TYPE ST_HIERARCHYDATALIST :
STRUCT
	TRACKINGLEVELS		:STRING;
	HIERARCHYDATAPK		:STRING;
	HIERARCHYDATAOUT	:STRING;
	HIERARCHYDATACS		:STRING;
END_STRUCT
END_TYPE

(* stored: Version 1.1.0.1, ProductVersion 3.1.4024.13
   DUT ST_HIERARCHYDATALIST: Id {e0bf9814-02fe-40a9-a2f4-09508059ba4f} *)
